// Block: A0302_Bordatrice_RegolazioneFormato_PERS

DATA_BLOCK A0302_Bordatrice_RegolazioneFormato_PERS
VERSION : 0.1
   NON_RETAIN
   VAR
      Par_Machine : Struct
         Nervatura_Pos_Riposo : Real;
         Passaggio01_MaxDisallineamentoAXs : Real;
         Passaggio02_MaxDisallineamentoAXs : Real;
         Passaggio03_MaxDisallineamentoAXs : Real;
         Passaggio04_MaxDisallineamentoAXs : Real;
         AxD_AutoSpeed : Real;
      END_STRUCT;
      Par_Enc : Array[1..9] of PosFbk_RTN;
      Par_D : Array[1..1] of Positioning_DOL_Machine_Par;
      Par_M : Array[2..9] of Positioning_MOL_Machine_Par;
      Pers_D : Array[1..1] of Positioning_DOL_Machine_Pers_Data;
      Pers_M : Array[2..9] of Positioning_MOL_Machine_Pers_Data;
   END_VAR

BEGIN
   // No initialization required
END_DATA_BLOCK
